(* IEC 61131-3 sources: ae-hw-engineering/src, 4 files *)

(* ---- cpu1516v31_IoAddresses.st ---- *)
CONFIGURATION IoAddresses

    VAR_GLOBAL
        et200s_device_di2_1_InputAddress AT %IB1: BYTE;
        et200s_device_di2_2_InputAddress AT %IB0: BYTE;
        et200s_device_dq2_1_OutputAddress AT %QB1: BYTE;
        et200s_device_dq2_2_OutputAddress AT %QB0: BYTE;
        et200sp1_device_di8_InputAddress AT %IB3: BYTE;
        et200sp1_device_dq8_OutputAddress AT %QB3: BYTE;
        et200sp2_device_di8_InputAddress AT %IB2: BYTE;
        et200sp2_device_dq8_OutputAddress AT %QB2: BYTE;
    END_VAR

END_CONFIGURATION

(* ---- configuration.st ---- *)
CONFIGURATION MyConfiguration
    TASK Main(Interval := T#1000ms, Priority := 1);
    PROGRAM P1 WITH Main: MainProgram;

    VAR_GLOBAL
        et200s_device_2DI_1_InputAddress AT %IB1: BYTE;
        et200s_device_2DI_2_InputAddress AT %IB0: BYTE;
        et200s_device_2DQ_1_OutputAddress AT %QB0: BYTE;
        et200s_device_2DQ_2_OutputAddress AT %QB66: BYTE;
        et200sp1_device_di8_InputAddress AT %IB3: BYTE;
        et200sp1_device_dq8_OutputAddress AT %QB2: BYTE;
        et200sp2_device_di8_InputAddress AT %IB2: BYTE;
        et200sp2_device_dq8_OutputAddress AT %QB1: BYTE;

        {S7.extern=ReadWrite}
        {OpcUA = ReadWrite}
        set_output : BOOL;
    END_VAR
END_CONFIGURATION

(* ---- MainProgram.st ---- *)
PROGRAM MainProgram

    VAR_EXTERNAL
        et200sp1_device_dq8_OutputAddress : BYTE;
        et200sp2_device_dq8_OutputAddress : BYTE;
        set_output : BOOL;
    END_VAR
    VAR
        counter : INT := 0;
    END_VAR

    counter := counter + 1;
    IF counter > 255 THEN
        counter := 0;
    END_IF;

    // set each output of the signal module "device_dq8" plugged to the IO device "et200sp1_device"
    et200sp1_device_dq8_OutputAddress := TO_BYTE(counter);

    // set the output 0 of the signal module "device_dq8" plugged to the IO device "et200sp2_device" depending on the variable set_output which can be controlled via OPC UA or Web Server
    et200sp2_device_dq8_OutputAddress.%X0 := set_output;

END_PROGRAM

(* ---- program.st ---- *)
PROGRAM MyProgram
    VAR_EXTERNAL
        et200sp1_device_dq8_OutputAddress : BYTE;
        et200sp2_device_dq8_OutputAddress : BYTE;
        set_output : BOOL;
    END_VAR
    VAR
        counter : INT := 0;
    END_VAR
    VAR_TEMP
    END_VAR
    counter := counter + 1;
    IF counter > 255 THEN
        counter := 0;
    END_IF;

    // set each output of the signal module "device_dq8" plugged to the IO device "et200sp1_device"
    et200sp1_device_dq8_OutputAddress := TO_BYTE(counter);

    // set the output 0 of the signal module "device_dq8" plugged to the IO device "et200sp2_device" depending on the variable set_output which can be controlled via OPC UA or Web Server
    et200sp2_device_dq8_OutputAddress.%X0 := set_output;

END_PROGRAM
